(* CoDeSys 2.3 export: GetStringLengthMax.EXP *)

(* POU MQTT-Utils/GetStringLengthMax, ST *)
FUNCTION GetStringLengthMax : UINT
VAR_INPUT
	pString			: POINTER TO BYTE;
	MaxLength		: UINT;
END_VAR
VAR
END_VAR
GetStringLengthMax := 0;
WHILE pString^ <> 0 AND GetStringLengthMax < MaxLength DO
	pString := pString + 1;
	GetStringLengthMax := GetStringLengthMax + 1;
END_WHILE
END_FUNCTION
